FUNCTION_BLOCK CommandBuffer
VAR_INPUT
END_VAR
VAR_OUTPUT
END_VAR
VAR
	commandArray : ARRAY [0..MAX_ENTRIES] OF I_Command;
	lastIndex : INT := EMPTY;
	emptyCommand : CommandNull;
END_VAR
VAR CONSTANT
	EMPTY : INT := -1;
	MAX_ENTRIES : INT := 10;
	FIRST_ENTRY : INT := 0;
	LAST_ENTRY : INT := MAX_ENTRIES -1;
END_VAR

PROPERTY PUBLIC CurrentCommand : I_Command
GET
IF isEmpty THEN
	CurrentCommand := emptyCommand;
ELSE 
	CurrentCommand := commandArray[FIRST_ENTRY];
END_IF
END_GET
END_PROPERTY

METHOD PUBLIC Insert : BOOL
VAR_INPUT
	cmd : I_Command;
END_VAR
IF isFull THEN
	RETURN;
END_IF

lastIndex := lastIndex + 1;
commandArray[lastIndex] := cmd;
Insert := TRUE;
END_METHOD

PROPERTY PUBLIC isEmpty : BOOL
GET
isEmpty := (lastIndex = EMPTY);
END_GET
END_PROPERTY

PROPERTY PUBLIC isFull : BOOL
GET
isFull := (lastIndex = MAX_ENTRIES);
END_GET
END_PROPERTY

METHOD PUBLIC Next
VAR_INPUT
END_VAR
IF isEmpty THEN
	RETURN;
END_IF

Shift();
END_METHOD

METHOD PRIVATE Shift
VAR_INPUT
END_VAR
VAR
	i: INT;
END_VAR
commandArray[FIRST_ENTRY].Destroy();

FOR i := 1 TO lastIndex + 1 DO
	commandArray[i-1] := commandArray[i];
END_FOR

lastIndex := lastIndex - 1;
END_METHOD

END_FUNCTION_BLOCK

(* stored: Version 1.1.0.1, ProductVersion 3.1.4024.9
   POU CommandBuffer: Id {fb835ec9-ebc0-4252-93e9-37c3088632da}, SpecialFunc None
   Property CurrentCommand: Id {dcbb658b-8616-4d34-bf5d-6e9e277e4d67}
   Get Get: Id {082c7f55-ca65-454a-a19d-81415d311401}
   Method Insert: Id {b0881e18-d3be-43a9-a387-06533c1edd4a}
   Property isEmpty: Id {b39a5568-4f58-4ad2-a30a-194dad8dc0f8}
   Get Get: Id {a5cc405d-90d4-4967-a569-eb1c56116337}
   Property isFull: Id {ffee4067-6051-4d22-9503-ad3598cfbd35}
   Get Get: Id {c3c50f92-093a-4edd-8e72-0254a9b5084b}
   Method Next: Id {6ee872c8-f5f6-4fe2-ae99-a5161c824e4b}
   Method Shift: Id {2b523c92-3515-4c3b-8688-5e8d7e910d4c} *)
